{attribute 'qualified_only'}
{attribute 'strict'}
TYPE E_System_Mode :
(
	System_Init := 0,
	System_Run

);
END_TYPE

(* stored: Version 1.1.0.1, ProductVersion 3.1.4024.9
   DUT E_System_Mode: Id {023219b4-3d19-4731-b642-8f3583dbae0b} *)
